FUNCTION_BLOCK E_REND (* Rendezvous of two events *)
  (* Standard: 61499-1-A; Classification: Event Processing *)
  (* Version 0.1, 2001-09-18, JHC, Rockwell Automation, XML version *)
  (* Version 0.0, 1996-11-22, JHC, Rockwell Automation, SRC version *)
  (* Compiler header: package fb.rt.events; *)
  (* Compiler Java IBM VisualAge 3.0 *)
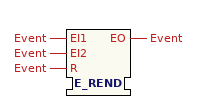
  EVENT_INPUT
    EI1; (* First Event Input *)
    EI2; (* Second Event Input *)
    R; (* Reset Event *)
  END_EVENT
  EVENT_OUTPUT
    EO; (* Rendezvous Output Event *)
  END_EVENT
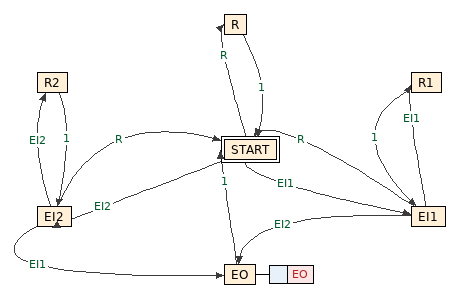
  EC_STATES
    START; (* Initial State *)
    R; (* Do nothing if R arrives when not awaiting rendezvous *)
    R1; (* Do nothing if EI1 arrives again while awaiting EI2 *)
    EI1; (* EI1 has arrived,wait for EI2 or R *)
    EO : -> EO; (* Issue rendezvous event *)
    EI2; (* EI2 has arrived,wait for EI1 or R *)
    R2; (* Do nothing if EI2 arrives again while awaiting EI1 *)
  END_STATES
  EC_TRANSITIONS
    START TO R := R;
    R TO START := 1;
    START TO EI1 := EI1;
    EI1 TO START := R;
    START TO EI2 := EI2;
    EI2 TO START := R;
    EI1 TO R1 := EI1;
    R1 TO EI1 := 1;
    EI2 TO R2 := EI2;
    R2 TO EI2 := 1;
    EI1 TO EO := EI2;
    EI2 TO EO := EI1;
    EO TO START := 1;
  END_TRANSITIONS
END_FUNCTION_BLOCK
